(* CoDeSys 2.3 export: FB_TOGGLE.EXP *)

(* POU FBs/FB_Toggle, ST *)
FUNCTION_BLOCK FB_Toggle
VAR_INPUT
	onTime: TIME :=  t#0.5s;
	offTime: TIME := t#1s;
END_VAR
VAR_OUTPUT
	Q: BOOL;
END_VAR
VAR
	t1: TON;
	t2: TOF;
END_VAR
t1(IN := NOT t2.Q, pt := offTime);
t2(IN := t1.Q, pt := onTime);
Q := t2.Q;
END_FUNCTION_BLOCK
